FUNCTION_BLOCK FB_ROB EXTENDS FB_Base IMPLEMENTS ITF_1_Robot

VAR_INPUT
	nErrorId : UINT; //FIX BUG
	PM: FB_PointManager;
// 	FILESERVER: FB_FileServer;
END_VAR


VAR_OUTPUT
    bCommunicationReady : BOOL;
    bReady : BOOL;
    bEnabled : BOOL;
    bMoving : BOOL;
    bBusy : BOOL;
    bInCollision : BOOL;
    eModus : eMode;
    
END_VAR

VAR
	_speedOverride : LREAL := 100.0;
	index: INT;
END_VAR

PROPERTY Busy : BOOL
GET
Busy := bBusy;
END_GET
SET
bBusy := Busy;
END_SET
END_PROPERTY

PROPERTY Collision : BOOL
GET
Collision := bInCollision;
END_GET
END_PROPERTY

PROPERTY CommunicationReady : BOOL
GET
// CommunicationReady := FB_ROB.bCommunicationReady;
END_GET
SET
// FB_ROB.bCommunicationReady := CommunicationReady;
END_SET
END_PROPERTY

ACTION CYCLIC_ROB:
CYCLIC_BASE();

FOR index := TO_INT(LOWER_BOUND(pA_Skills, 1)) TO TO_INT(UPPER_BOUND(pA_Skills, 1)) DO
    IF pA_Skills[index] <> 0 THEN
        pA_Skills[index]^.StateMachine();
    END_IF
END_FOR


PM();
END_ACTION

METHOD DisableRobot : BOOL
bEnabled := FALSE;
DisableRobot := Deactivate();
END_METHOD

METHOD EnableRobot : BOOL
bEnabled := TRUE;
EnableRobot := TRUE;
END_METHOD

PROPERTY Mode : eMode
GET
Mode := eModus;
END_GET
SET
eModus := Mode;
END_SET
END_PROPERTY

METHOD PROTECTED OnActivate : eResult
eModus := eMode.Automatic;
OnActivate := eResult.SUCCESS;
END_METHOD

METHOD PROTECTED OnCleanup : eResult
END_METHOD

METHOD PROTECTED OnConfigure : eResult
// ---- Init ----
_transitionresult := eResult.None;

// ---- Change ----
eModus := eMode.Manual;
// Connect();

// ---- Check ----
IF bError THEN
    _transitionresult := eResult.ERROR;
ELSIF CommunicationReady THEN
    _transitionresult := eResult.SUCCESS;
END_IF

// ---- Change State ----
OnConfigure := _transitionresult;
END_METHOD

METHOD PROTECTED OnDeactivate : eResult
eModus := eMode.Manual;
OnDeactivate := eResult.SUCCESS;
END_METHOD

METHOD PROTECTED OnError : eResult
eModus := eMode.Manual;
OnError := eResult.SUCCESS;
END_METHOD

METHOD PROTECTED OnShutdown : eResult
eModus := eMode.Manual;
OnShutdown := eResult.SUCCESS;
END_METHOD

METHOD Pause : BOOL
Pause := FALSE;
END_METHOD

METHOD ResetRobot : BOOL
bError := FALSE;
nErrorId := 0;
ResetRobot := TRUE;
END_METHOD

METHOD Resume : BOOL
Resume := FALSE;
END_METHOD

PROPERTY RobotEnabled : BOOL
GET
RobotEnabled := bEnabled;
END_GET
SET
bEnabled := RobotEnabled;
END_SET
END_PROPERTY

PROPERTY RobotError : BOOL
GET
RobotError := bError;
END_GET
END_PROPERTY

PROPERTY RobotMoving : BOOL
GET
RobotMoving := bMoving;
END_GET
SET
bMoving := RobotMoving;
END_SET
END_PROPERTY

PROPERTY RobotReady : BOOL
GET
RobotReady := bReady;
END_GET
SET
bReady := RobotReady;
END_SET
END_PROPERTY

METHOD SetOperationMode : BOOL
VAR_INPUT
    mode : eMode;
END_VAR
eModus := mode;
SetOperationMode := TRUE;
END_METHOD

METHOD SetSpeedOverride : BOOL
VAR_INPUT
    factor : LREAL;
END_VAR
IF (factor < 0.001) OR (factor > 100.0) THEN
    SetSpeedOverride := FALSE;
    RETURN;
END_IF
_speedOverride := factor;
SetSpeedOverride := TRUE;
END_METHOD

METHOD Stop : BOOL
Stop := FALSE;
END_METHOD

END_FUNCTION_BLOCK

(* stored: Version 1.1.0.1, ProductVersion 3.1.4026.18
   POU FB_ROB: Id {7ce28b50-28f8-4d4c-bb25-1006bf064637}, SpecialFunc None
   Folder Generic Control: Id {d269719e-4481-455b-8abd-a0a346547cd3}
   Folder Generic Motion Settings: Id {e84a80be-ec15-4bef-9f1f-3428dddc27ab}
   Folder Generic Status: Id {c1e8e35a-1828-4d72-a2cb-3aa1cc7ab721}
   Folder StateControl: Id {306f9b72-2cb2-4dec-88a3-0a1776eb8cb9}
   Property Busy: Id {9cc952da-997b-48e1-bc3f-e76175b74970}
   Get Get: Id {19a4579d-a5c4-4a8f-b588-1cda29eef266}
   Set Set: Id {2c85e6a2-337f-449c-aad2-4b015e26ecdd}
   Property Collision: Id {8eea56b9-50ca-4510-b567-db19e3eca5c7}
   Get Get: Id {885867df-c0d3-4443-aec9-8d2b982d6c40}
   Property CommunicationReady: Id {80fca5f5-8709-4982-a384-df957ec0f13e}
   Get Get: Id {99f48d79-5a32-4dfc-8ac6-28f7e421e088}
   Set Set: Id {a3a4030b-8d2a-45fa-89c6-94fd0d2368eb}
   Action CYCLIC_ROB: Id {ebf16c89-c511-406b-9426-1ade99c4f730}
   Method DisableRobot: Id {bbb8a1cb-19df-48a2-aa34-15efcd08818d}
   Method EnableRobot: Id {3bb80d4c-ff29-49a1-abc5-c8b4d3120296}
   Property Mode: Id {b02ce28c-7dc7-4355-aadb-75f0e04880fa}
   Get Get: Id {5422baec-3cfa-49de-a9e5-c204b5dc3b85}
   Set Set: Id {70edccef-4005-4ebc-8367-68039a4d1e15}
   Method OnActivate: Id {92a2cf27-c6ee-447f-b5b4-e372093c0834}
   Method OnCleanup: Id {b8d25f1a-bd56-4d52-bf77-294e7c965601}
   Method OnConfigure: Id {fb57d4c1-8d73-4b61-a93c-ea33b423e3bc}
   Method OnDeactivate: Id {9cfadd55-1f96-401b-82a9-c49bdb0b9d71}
   Method OnError: Id {af5714ff-685b-4718-92d7-e4e00300345c}
   Method OnShutdown: Id {54edc0cd-8c64-49fa-9d9a-b9e92650f21c}
   Method Pause: Id {4e031858-9871-4cbe-80c4-7b945008a9d5}
   Method ResetRobot: Id {3ea33c07-baa7-444c-a0bc-e71071e519dd}
   Method Resume: Id {5d4cc18a-f3ec-4e77-a0a2-63e6b1c4f8da}
   Property RobotEnabled: Id {8b95af0d-0de5-4e03-a42f-b367f7d60c51}
   Get Get: Id {e7fba8f0-0b85-4bb7-b5f5-3bbf4b89f164}
   Set Set: Id {d9bda0f1-a1cd-4d1c-9f6d-88ca4e5d9cc1}
   Property RobotError: Id {e8095074-bc2d-49ad-8f7a-7a4d7677a8f7}
   Get Get: Id {25903a36-625c-4391-b5b1-be1d7b80d6fa}
   Property RobotMoving: Id {35ca0c87-c7ee-4f80-a87b-f8e0bf6781ef}
   Get Get: Id {4af7c180-96b4-478d-9ba7-15a9132d033d}
   Set Set: Id {8c3ef50b-f0bb-4f67-b971-f8d926a0360c}
   Property RobotReady: Id {8f2c7f81-6dd1-4fa4-9c6b-42ea40f162a7}
   Get Get: Id {64b31d92-9d68-4b99-8d36-01a37d3c1eb9}
   Set Set: Id {1b0d1b5e-b5d6-42fc-b350-c4d2c9dd5ba9}
   Method SetOperationMode: Id {a36cbff6-922e-4670-8cae-63446b6e1765}
   Method SetSpeedOverride: Id {a5e39256-a687-447d-8a2a-a95ea9e40d2e}
   Method Stop: Id {ff1c583d-626a-4142-b727-591a7a8cf9e6} *)
